(* PLC project Tc2_Utilities.LREAL_TO_INT64 Demo, tc3-libraries-kb TwinCAT 3.1 *)
(* stored: creationDateTime 2026-05-10T17:00:00, modificationDateTime 2026-05-10T17:00:00 *)

PROGRAM P_Demo_LREAL_TO_INT64
  VAR
    rResult : T_LARGE_INTEGER;  (* LREAL_TO_INT64 返回值 *)
    bRun : BOOL;  (* 触发一次调用 *)
    rX : LREAL := 1.234E9;  (* 测试用本地变量 *)
  END_VAR

            // ============================================================
// Tc2_Utilities.LREAL_TO_INT64 演示程序（FUNCTION）
// ============================================================
// 验证步骤：
//   1. 引用 Tc2_Utilities
//   2. 编译 + 登录
//   3. 强制 bRun := TRUE 一个周期
//   4. 在线监视 rResult
// ============================================================

IF bRun THEN
    rResult := LREAL_TO_INT64(rX);
    bRun := FALSE;
END_IF;

          
END_PROGRAM
